Staubli VAL3: extractRows.pgx

public program extractRows(num& x_nInput[] (dimensions=2), num& x_nIndices[], num& x_nResult[] (dimensions=2))
  local num l_nCol
  local num l_nCounter
  local num l_nRow
begin

  resize(x_nResult,1,1)
  resize(x_nResult,2,1)
  x_nResult[0,0] = 0
  resize(x_nResult,1, size(x_nIndices))
  resize(x_nResult,2, size(x_nInput,2))

  for l_nRow = 0 to size(x_nIndices)-1
    for l_nCol = 0 to size(x_nInput,2)-1
      x_nResult[l_nRow, l_nCol] = x_nInput[x_nIndices[l_nRow],l_nCol]
    endFor
  endFor

end
